TEXTLIST TextList_Arm_Setting
  1 = '1'
  2 = '2'
  3 = '3'
  4 = '4'
  5 = '5'
  6 = '6'
  7 = 'LOADING'
  8 = 'UNLOADING'
   = ''
END_TEXTLIST

(* stored: Version 1.1.0.1, ProductVersion 3.1.4024.12
   TextList TextList_Arm_Setting: Id {24a3a443-2c2a-4621-b80c-49327c1bd86a} *)
